(* Logix 5000 project; controller Safety vendor 1 type 14 code 86 rev 19.11; software revision 19.01; part 7 of 17 *)
(* tags used below, declared in another part *)
   ToCitect4 : DINT[64];   // (To Citect4)
   x172CR460 : ALIAS FOR SDPLC:1:I.Pt00Data;   // Shear Die Drive Main Contactor Safety Relay Input
   x172CR510 : ALIAS FOR SDPLC:1:I.Pt01Data;   // Shear Die Drive Enable Safety Relay Input
   x533PB470a : ALIAS FOR H1:6:I.Pt00Data;   // Sheeter Emergency Stop Pushbutton
   x533PB470b : ALIAS FOR H1:6:I.Pt01Data;   // Sheeter Emergency Stop Pushbutton
   x702MTR191FF : ALIAS FOR MCC1:1:I.Pt00Data;   // Rewind Pinch Roll Fwd Fdbk
   x702MTR191RF : ALIAS FOR MCC1:1:I.Pt01Data;   // Rewind Pinch Roll Rev Fdbk
   x708MTR080FF : ALIAS FOR MCC1:1:I.Pt04Data;   // Flattener Drive Motor Fwd Fdbk
   x708MTR080RF : ALIAS FOR MCC1:1:I.Pt05Data;   // Flattener Drive Motor Rev Fdbk
   x708MTR250FF : ALIAS FOR MCC1:1:I.Pt06Data;   // Unwind Holddown Roll Drive Motor Fwd Fdbk
   x708MTR250RF : ALIAS FOR MCC1:1:I.Pt07Data;   // Unwind Holddown Roll Drive Motor Rev Fdbk
   x753MTR190FF : ALIAS FOR MCC3:1:I.Pt00Data;   // Trimmer Pinch Roll Fwd Fdbk
   x753MTR190RF : ALIAS FOR MCC3:1:I.Pt01Data;   // Trimmer Pinch Roll Rev Fdbk
   x759MTR080SE : ALIAS FOR MCC3:4:O.Pt02Data;   // Scrap Choppers Width Adjust Safety Enable
   x759MTR080SP : ALIAS FOR MCC3:4:O.Pt01Data;   // Scrap Choppers Width Adjust Safety Power
   x761MTR081RF : ALIAS FOR MCC3:1:I.Pt02Data;   // Trimmer Scrap Conveyor RunFdbk
   x778MTR080RF : ALIAS FOR MCC4:1:I.Pt00Data;   // Shear Crank Motor Run Fdbk
   x802MTR080FF : ALIAS FOR MCC5:1:I.Pt00Data;   // Stacker Side Guide Lift Fwd Fdbk/Up
   x802MTR080RF : ALIAS FOR MCC5:1:I.Pt01Data;   // Stacker Side Guide Lift Rev Fdbk/Down
   x802MTR230FF : ALIAS FOR MCC5:1:I.Pt02Data;   // Scrap Horizontal Conveyor Run Fwd Fdbk
   x802MTR230RF : ALIAS FOR MCC5:1:I.Pt03Data;   // Scrap Horizontal Conveyor Run Rev Fdbk
   x802MTR231FF : ALIAS FOR MCC5:1:I.Pt04Data;   // Stacker Chain Fwd Fdbk
   x802MTR231RF : ALIAS FOR MCC5:1:I.Pt05Data;   // Stacker Chain Rev Fdbk
   y172CR460 : ALIAS FOR SDPLC:2:O.Pt00Data;   // Shear Die Drive Main Contactor Safety Relay Output
   y172CR510 : ALIAS FOR SDPLC:2:O.Pt01Data;   // Shear Die Drive Enable Safety Relay Output
   y172CR550 : ALIAS FOR SDPLC:2:O.Pt02Data;   // Line Soleniod Safe-Off
   y702MTR191FC : ALIAS FOR MCC1:6:O.Pt00Data;   // Rewind Pinch Roll Fwd Cmd
   y702MTR191RC : ALIAS FOR MCC1:6:O.Pt01Data;   // Rewind Pinch Roll Rev Cmd
   y708MTR080FC : ALIAS FOR MCC1:6:O.Pt04Data;   // Flattener Drive Motor Fwd Cmd
   y708MTR080RC : ALIAS FOR MCC1:6:O.Pt05Data;   // Flattener Drive Motor Rev Cmd
   y708MTR250FC : ALIAS FOR MCC1:6:O.Pt06Data;   // Unwind Holddown Roll Drive Motor Fwd Cmd
   y708MTR250RC : ALIAS FOR MCC1:6:O.Pt07Data;   // Unwind Holddown Roll Drive Motor Rev Cmd
   y725MTR080SE : ALIAS FOR MCC2:1:O.Pt01Data;   // Unwind Pinch Roll Safety Enable
   y725MTR080SP : ALIAS FOR MCC2:1:O.Pt00Data;   // Unwind Pinch Roll Safety Power
   y727MTR080SE : ALIAS FOR MCC2:1:O.Pt05Data;   // Paper Winder Safety Enable
   y727MTR080SP : ALIAS FOR MCC2:1:O.Pt04Data;   // Paper Winder Safety Power
   y729MTR080SE : ALIAS FOR MCC2:1:O.Pt03Data;   // Washtank Pinch Roll 4 Safety Enable
   y729MTR080SP : ALIAS FOR MCC2:1:O.Pt02Data;   // Washtank Pinch Roll 4 Safety Power
   y731MTR080SE : ALIAS FOR MCC2:1:O.Pt07Data;   // Washtank Pinch Roll 1 Safety Enable
   y731MTR080SP : ALIAS FOR MCC2:1:O.Pt06Data;   // Washtank Pinch Roll 1 Safety Power
   y733MTR080SE : ALIAS FOR MCC2:2:O.Pt01Data;   // Washtank Pinch Roll 2 Safety Enable
   y733MTR080SP : ALIAS FOR MCC2:2:O.Pt00Data;   // Washtank Pinch Roll 2 Safety Power
   y735MTR080SE : ALIAS FOR MCC2:2:O.Pt03Data;   // Washtank Pinch Roll 3 Safety Enable
   y735MTR080SP : ALIAS FOR MCC2:2:O.Pt02Data;   // Washtank Pinch Roll 3 Safety Power
   y751MTR080SE : ALIAS FOR MCC3:3:O.Pt04Data;   // Trimmer Knives Safety Enable
   y751MTR080SP : ALIAS FOR MCC3:3:O.Pt03Data;   // Trimmer Knives Safety Power
   y753MTR190FC : ALIAS FOR MCC3:3:O.Pt00Data;   // Trimmer Pinch Roll Fwd Cmd
   y753MTR190RC : ALIAS FOR MCC3:3:O.Pt01Data;   // Trimmer Pinch Roll Rev Cmd
   y754MTR080SE : ALIAS FOR MCC3:3:O.Pt06Data;   // Side Guide Width Adjust Safety Enable
   y754MTR080SP : ALIAS FOR MCC3:3:O.Pt05Data;   // Side Guide Width Adjust Safety Power
   y755MTR080SE : ALIAS FOR MCC3:4:O.Pt00Data;   // Trimmer Knives Width Adjust Safety Enable
   y755MTR080SP : ALIAS FOR MCC3:3:O.Pt07Data;   // Trimmer Knives Width Adjust Safety Power
   y761MTR081RC : ALIAS FOR MCC3:3:O.Pt02Data;   // Trimmer Scrap Conveyor RunCmd
   y762MTR080SE : ALIAS FOR MCC3:4:O.Pt04Data;   // Scrap Choppers Safety Enable
   y762MTR080SP : ALIAS FOR MCC3:4:O.Pt03Data;   // Scrap Choppers Safety Power
   y776MTR080SE : ALIAS FOR MCC4:3:O.Pt07Data;   // Shear Metering Backup Roll Safety Enable
   y776MTR080SP : ALIAS FOR MCC4:3:O.Pt06Data;   // Shear Metering Backup Roll Safety Power
   y778MTR080RC : ALIAS FOR MCC4:4:O.Pt00Data;   // Shear Die Crank Run Cmd
   y779MTR080SE : ALIAS FOR MCC4:3:O.Pt01Data;   // Shear Pinch Roll Safety Enable
   y779MTR080SP : ALIAS FOR MCC4:3:O.Pt00Data;   // Shear Pinch Roll Safety Power
   y782MTR080SE : ALIAS FOR MCC4:3:O.Pt03Data;   // Sheeter Pinch Roll Safety Enable
   y782MTR080SP : ALIAS FOR MCC4:3:O.Pt02Data;   // Sheeter Pinch Roll Safety Power
   y785MTR080SE : ALIAS FOR MCC4:3:O.Pt05Data;   // Stacker Blower Safety Enable
   y785MTR080SP : ALIAS FOR MCC4:3:O.Pt04Data;   // Stacker Blower Safety Power
   y800MTR080SE : ALIAS FOR MCC5:3:O.Pt01Data;   // Scrap Incline Conveyor Safety Enable
   y800MTR080SP : ALIAS FOR MCC5:3:O.Pt00Data;   // Scrap Incline Conveyor Safety Power
   y802MTR080FC : ALIAS FOR MCC5:4:O.Pt04Data;   // Stacker Side Guide Lift Fwd Cmd/Up
   y802MTR080RC : ALIAS FOR MCC5:4:O.Pt05Data;   // Stacker Side Guide Lift Rev Cmd/Down
   y802MTR230FC : ALIAS FOR MCC5:4:O.Pt06Data;   // Scrap Horizontal Conveyor Fwd Cmd
   y802MTR230RC : ALIAS FOR MCC5:4:O.Pt07Data;   // Scrap Horizontal Conveyor Rev Cmd
   y802MTR231FC : ALIAS FOR MCC5:5:O.Pt00Data;   // Stacker Chain Fwd Cmd
   y802MTR231RC : ALIAS FOR MCC5:5:O.Pt01Data;   // Stacker Chain Rev Cmd
   y804MTR080SE : ALIAS FOR MCC5:3:O.Pt03Data;   // Stacker Back Stop Safety Enable
   y804MTR080SP : ALIAS FOR MCC5:3:O.Pt02Data;   // Stacker Back Stop Safety Power
   y806MTR080SE : ALIAS FOR MCC5:3:O.Pt05Data;   // Product Conveyor 3 Safety Enable
   y806MTR080SP : ALIAS FOR MCC5:3:O.Pt04Data;   // Product Conveyor 3 Safety Power
   y808MTR080SE : ALIAS FOR MCC5:3:O.Pt07Data;   // Product Conveyor 1 Safety Enable
   y808MTR080SP : ALIAS FOR MCC5:3:O.Pt06Data;   // Product Conveyor 1 Safety Power
   y810MTR080SE : ALIAS FOR MCC5:4:O.Pt01Data;   // Product Conveyor 2 Safety Enable
   y810MTR080SP : ALIAS FOR MCC5:4:O.Pt00Data;   // Product Conveyor 2 Safety Power
   y812MTR080SE : ALIAS FOR MCC5:4:O.Pt03Data;   // Shear Conveyor Safety Enable
   y812MTR080SP : ALIAS FOR MCC5:4:O.Pt02Data;   // Shear Conveyor Safety Power
(* Comms, continued *)

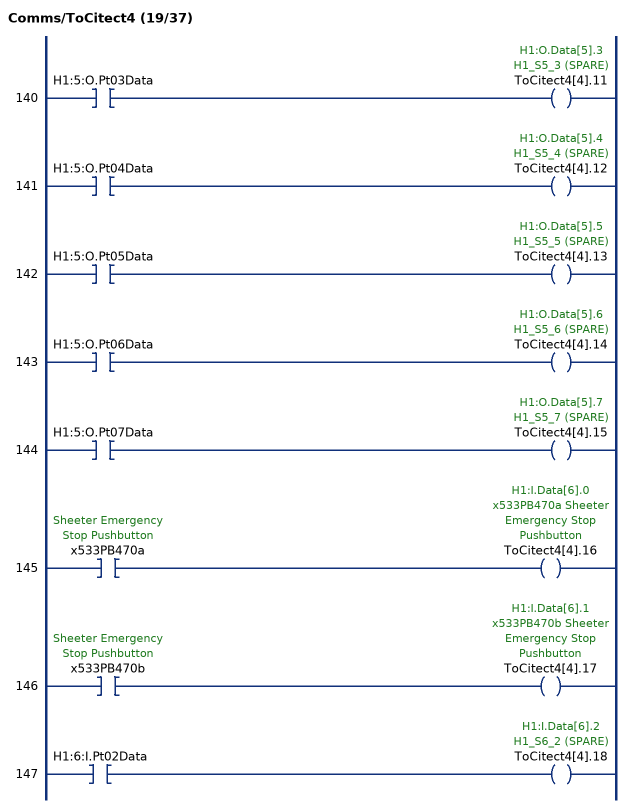
   140: XIC(H1:5:O.Pt03Data)OTE(ToCitect4[4].11);
   141: XIC(H1:5:O.Pt04Data)OTE(ToCitect4[4].12);
   142: XIC(H1:5:O.Pt05Data)OTE(ToCitect4[4].13);
   143: XIC(H1:5:O.Pt06Data)OTE(ToCitect4[4].14);
   144: XIC(H1:5:O.Pt07Data)OTE(ToCitect4[4].15);
   145: XIC(x533PB470a)OTE(ToCitect4[4].16);
   146: XIC(x533PB470b)OTE(ToCitect4[4].17);
   147: XIC(H1:6:I.Pt02Data)OTE(ToCitect4[4].18);
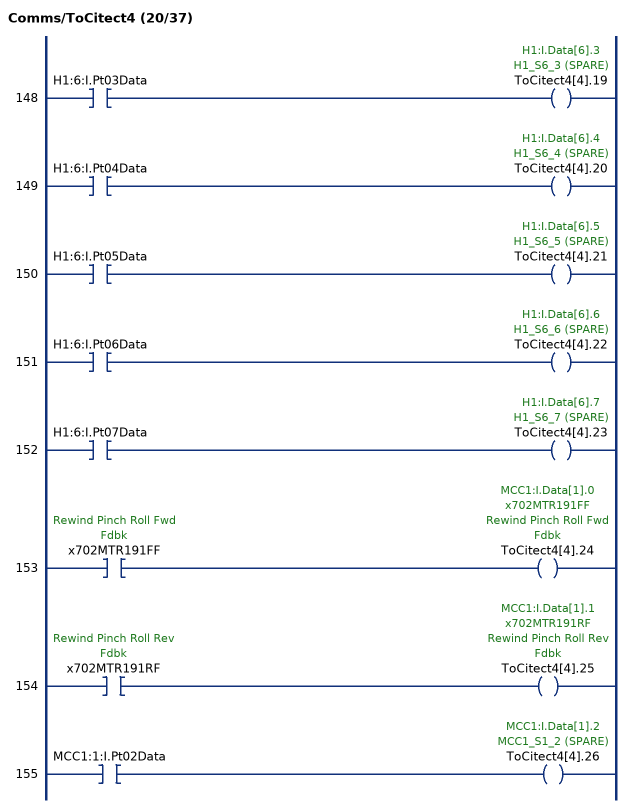
   148: XIC(H1:6:I.Pt03Data)OTE(ToCitect4[4].19);
   149: XIC(H1:6:I.Pt04Data)OTE(ToCitect4[4].20);
   150: XIC(H1:6:I.Pt05Data)OTE(ToCitect4[4].21);
   151: XIC(H1:6:I.Pt06Data)OTE(ToCitect4[4].22);
   152: XIC(H1:6:I.Pt07Data)OTE(ToCitect4[4].23);
   153: XIC(x702MTR191FF)OTE(ToCitect4[4].24);
   154: XIC(x702MTR191RF)OTE(ToCitect4[4].25);
   155: XIC(MCC1:1:I.Pt02Data)OTE(ToCitect4[4].26);
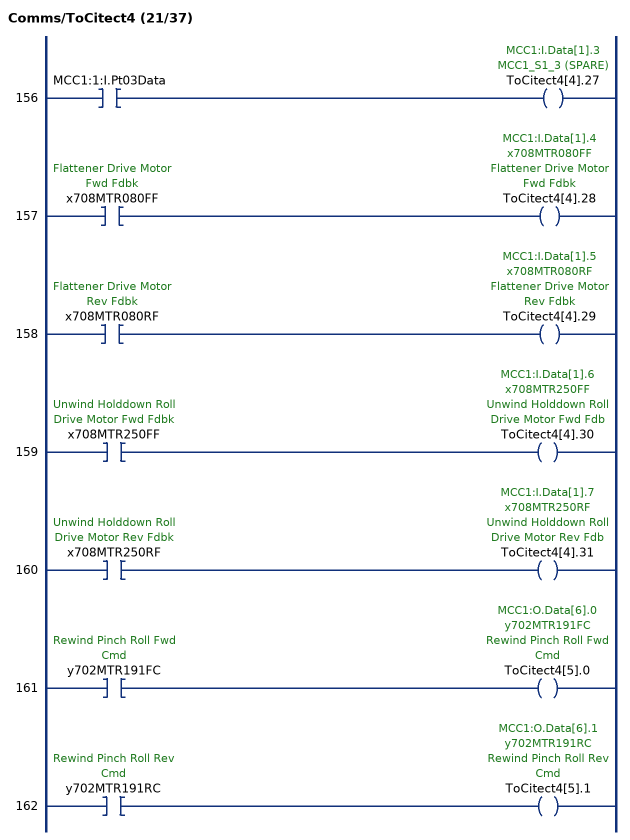
   156: XIC(MCC1:1:I.Pt03Data)OTE(ToCitect4[4].27);
   157: XIC(x708MTR080FF)OTE(ToCitect4[4].28);
   158: XIC(x708MTR080RF)OTE(ToCitect4[4].29);
   159: XIC(x708MTR250FF)OTE(ToCitect4[4].30);
   160: XIC(x708MTR250RF)OTE(ToCitect4[4].31);
   161: XIC(y702MTR191FC)OTE(ToCitect4[5].0);
   162: XIC(y702MTR191RC)OTE(ToCitect4[5].1);
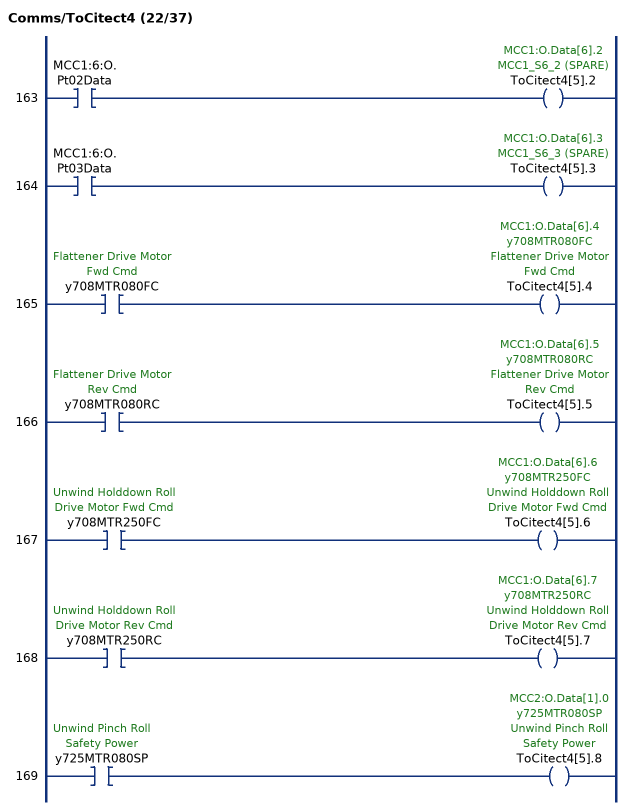
   163: XIC(MCC1:6:O.Pt02Data)OTE(ToCitect4[5].2);
   164: XIC(MCC1:6:O.Pt03Data)OTE(ToCitect4[5].3);
   165: XIC(y708MTR080FC)OTE(ToCitect4[5].4);
   166: XIC(y708MTR080RC)OTE(ToCitect4[5].5);
   167: XIC(y708MTR250FC)OTE(ToCitect4[5].6);
   168: XIC(y708MTR250RC)OTE(ToCitect4[5].7);
   169: XIC(y725MTR080SP)OTE(ToCitect4[5].8);
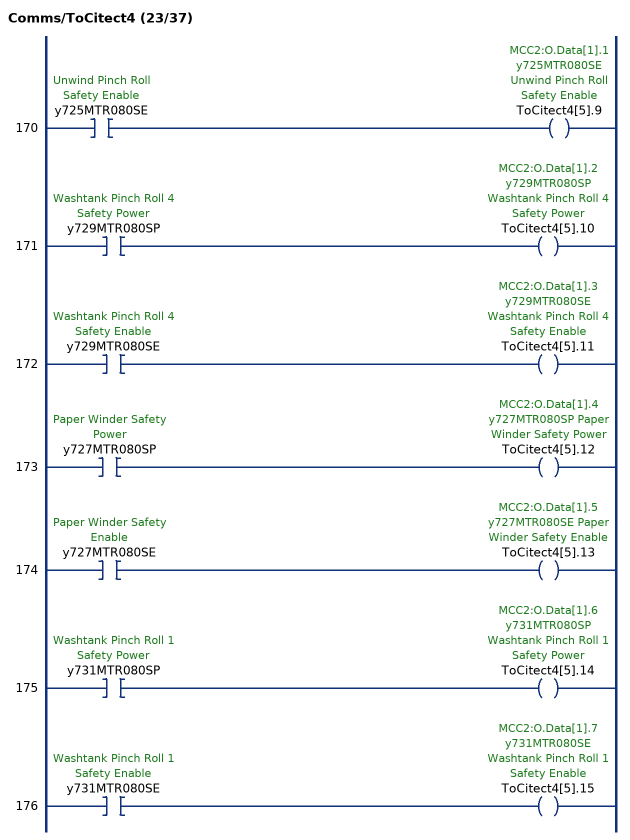
   170: XIC(y725MTR080SE)OTE(ToCitect4[5].9);
   171: XIC(y729MTR080SP)OTE(ToCitect4[5].10);
   172: XIC(y729MTR080SE)OTE(ToCitect4[5].11);
   173: XIC(y727MTR080SP)OTE(ToCitect4[5].12);
   174: XIC(y727MTR080SE)OTE(ToCitect4[5].13);
   175: XIC(y731MTR080SP)OTE(ToCitect4[5].14);
   176: XIC(y731MTR080SE)OTE(ToCitect4[5].15);
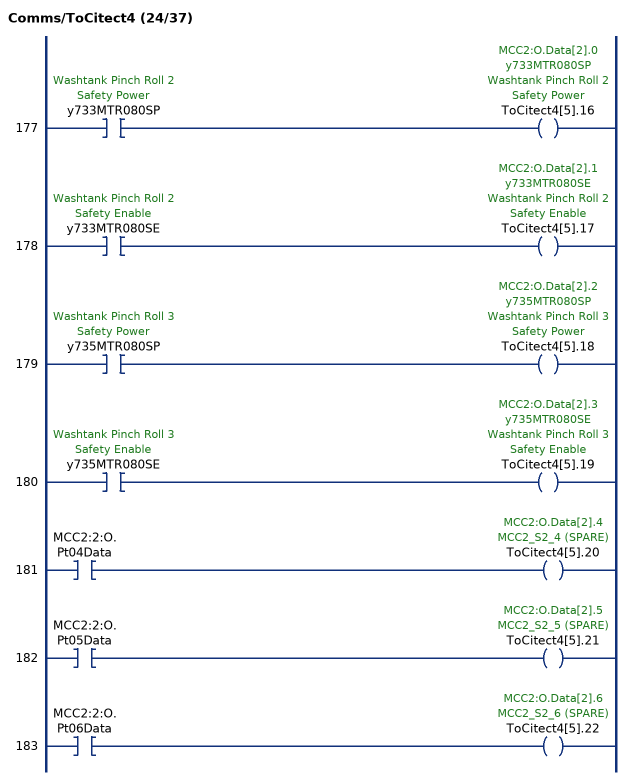
   177: XIC(y733MTR080SP)OTE(ToCitect4[5].16);
   178: XIC(y733MTR080SE)OTE(ToCitect4[5].17);
   179: XIC(y735MTR080SP)OTE(ToCitect4[5].18);
   180: XIC(y735MTR080SE)OTE(ToCitect4[5].19);
   181: XIC(MCC2:2:O.Pt04Data)OTE(ToCitect4[5].20);
   182: XIC(MCC2:2:O.Pt05Data)OTE(ToCitect4[5].21);
   183: XIC(MCC2:2:O.Pt06Data)OTE(ToCitect4[5].22);
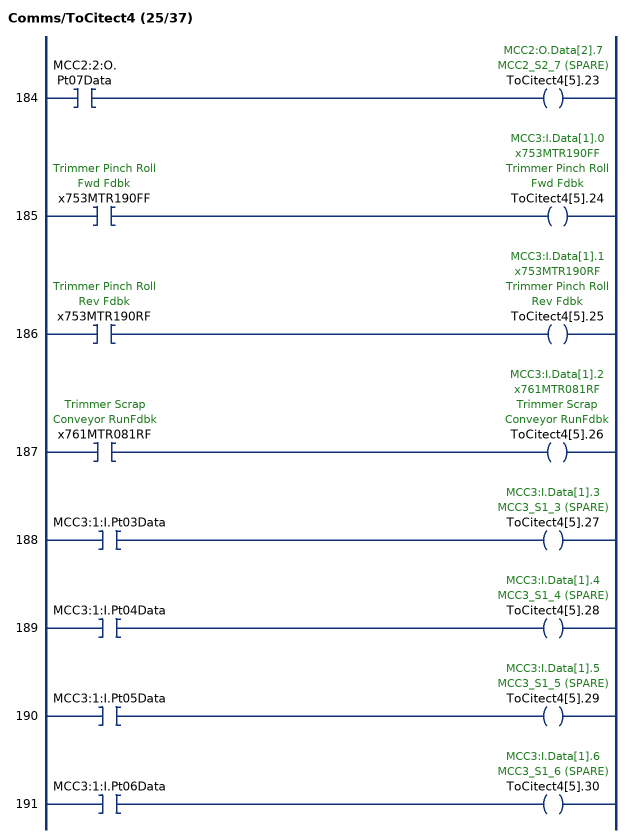
   184: XIC(MCC2:2:O.Pt07Data)OTE(ToCitect4[5].23);
   185: XIC(x753MTR190FF)OTE(ToCitect4[5].24);
   186: XIC(x753MTR190RF)OTE(ToCitect4[5].25);
   187: XIC(x761MTR081RF)OTE(ToCitect4[5].26);
   188: XIC(MCC3:1:I.Pt03Data)OTE(ToCitect4[5].27);
   189: XIC(MCC3:1:I.Pt04Data)OTE(ToCitect4[5].28);
   190: XIC(MCC3:1:I.Pt05Data)OTE(ToCitect4[5].29);
   191: XIC(MCC3:1:I.Pt06Data)OTE(ToCitect4[5].30);
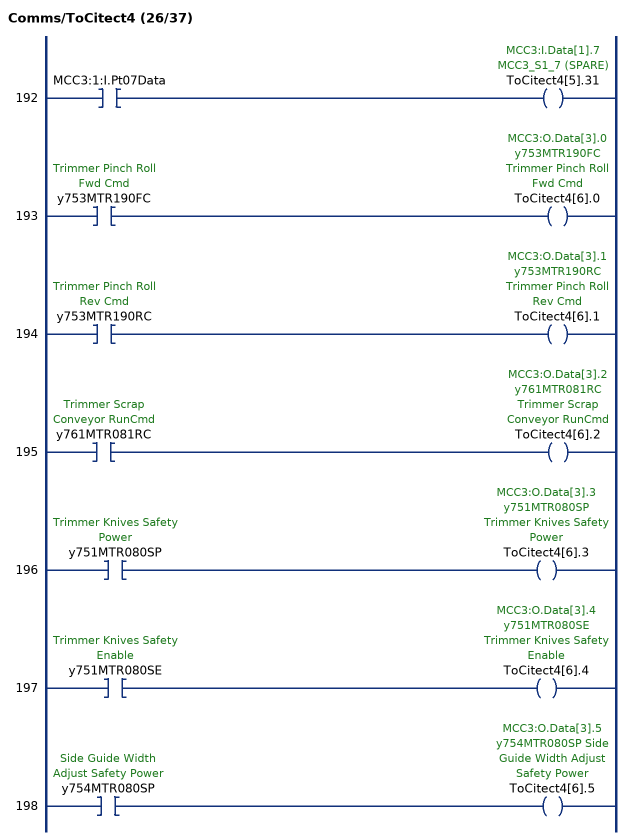
   192: XIC(MCC3:1:I.Pt07Data)OTE(ToCitect4[5].31);
   193: XIC(y753MTR190FC)OTE(ToCitect4[6].0);
   194: XIC(y753MTR190RC)OTE(ToCitect4[6].1);
   195: XIC(y761MTR081RC)OTE(ToCitect4[6].2);
   196: XIC(y751MTR080SP)OTE(ToCitect4[6].3);
   197: XIC(y751MTR080SE)OTE(ToCitect4[6].4);
   198: XIC(y754MTR080SP)OTE(ToCitect4[6].5);
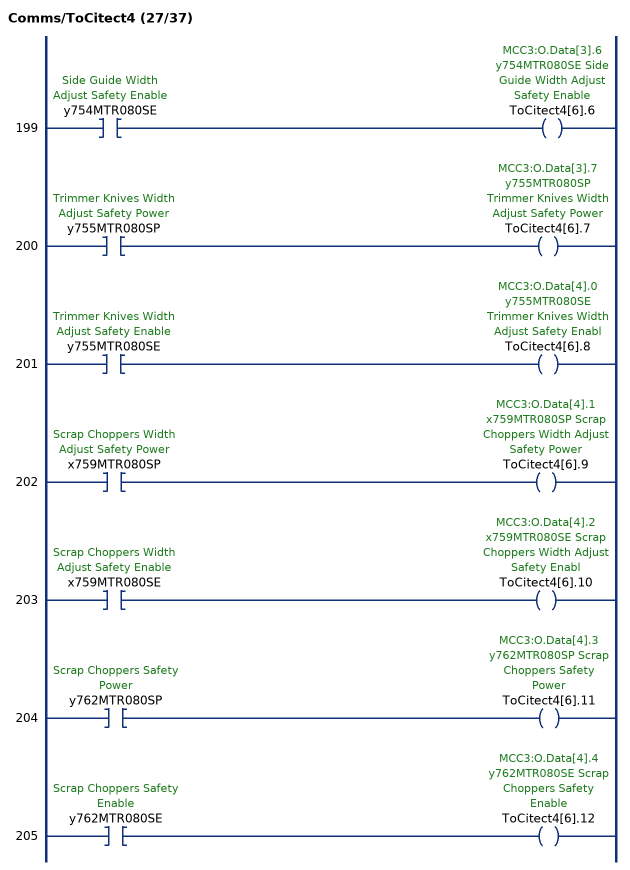
   199: XIC(y754MTR080SE)OTE(ToCitect4[6].6);
   200: XIC(y755MTR080SP)OTE(ToCitect4[6].7);
   201: XIC(y755MTR080SE)OTE(ToCitect4[6].8);
   202: XIC(x759MTR080SP)OTE(ToCitect4[6].9);
   203: XIC(x759MTR080SE)OTE(ToCitect4[6].10);
   204: XIC(y762MTR080SP)OTE(ToCitect4[6].11);
   205: XIC(y762MTR080SE)OTE(ToCitect4[6].12);
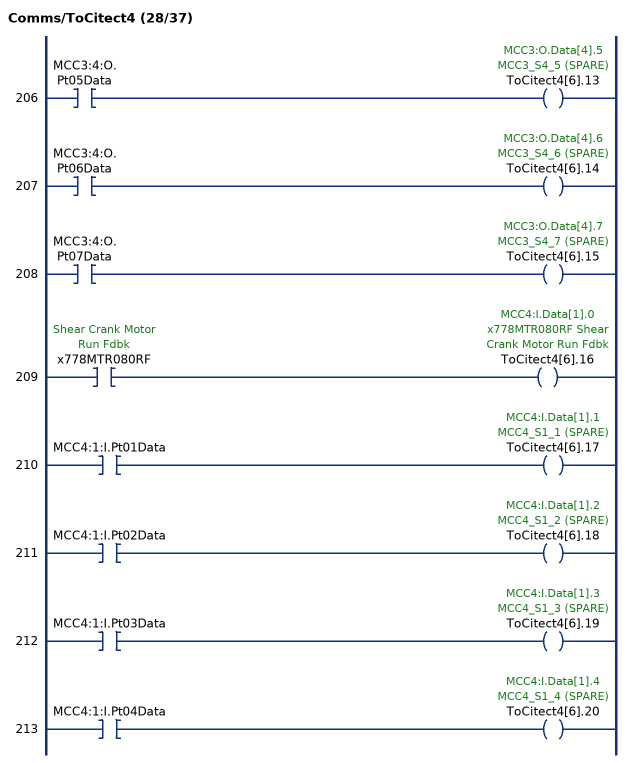
   206: XIC(MCC3:4:O.Pt05Data)OTE(ToCitect4[6].13);
   207: XIC(MCC3:4:O.Pt06Data)OTE(ToCitect4[6].14);
   208: XIC(MCC3:4:O.Pt07Data)OTE(ToCitect4[6].15);
   209: XIC(x778MTR080RF)OTE(ToCitect4[6].16);
   210: XIC(MCC4:1:I.Pt01Data)OTE(ToCitect4[6].17);
   211: XIC(MCC4:1:I.Pt02Data)OTE(ToCitect4[6].18);
   212: XIC(MCC4:1:I.Pt03Data)OTE(ToCitect4[6].19);
   213: XIC(MCC4:1:I.Pt04Data)OTE(ToCitect4[6].20);
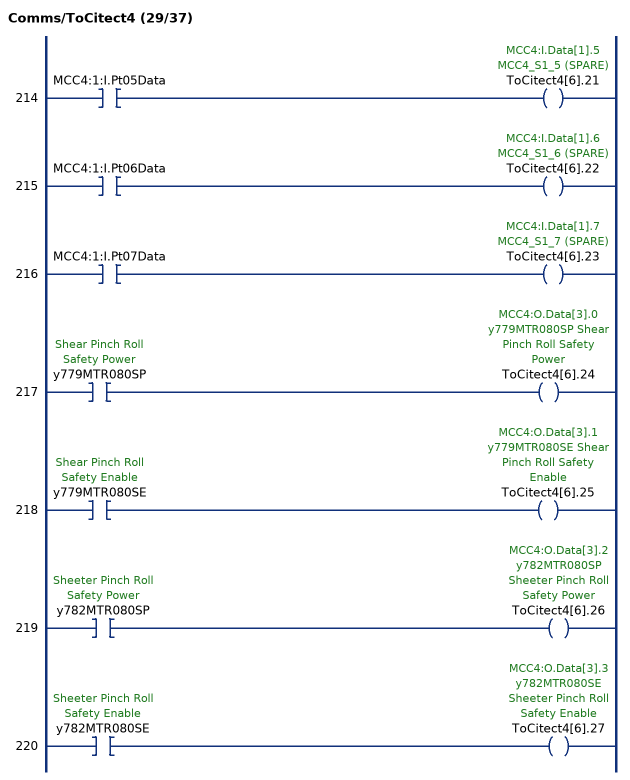
   214: XIC(MCC4:1:I.Pt05Data)OTE(ToCitect4[6].21);
   215: XIC(MCC4:1:I.Pt06Data)OTE(ToCitect4[6].22);
   216: XIC(MCC4:1:I.Pt07Data)OTE(ToCitect4[6].23);
   217: XIC(y779MTR080SP)OTE(ToCitect4[6].24);
   218: XIC(y779MTR080SE)OTE(ToCitect4[6].25);
   219: XIC(y782MTR080SP)OTE(ToCitect4[6].26);
   220: XIC(y782MTR080SE)OTE(ToCitect4[6].27);
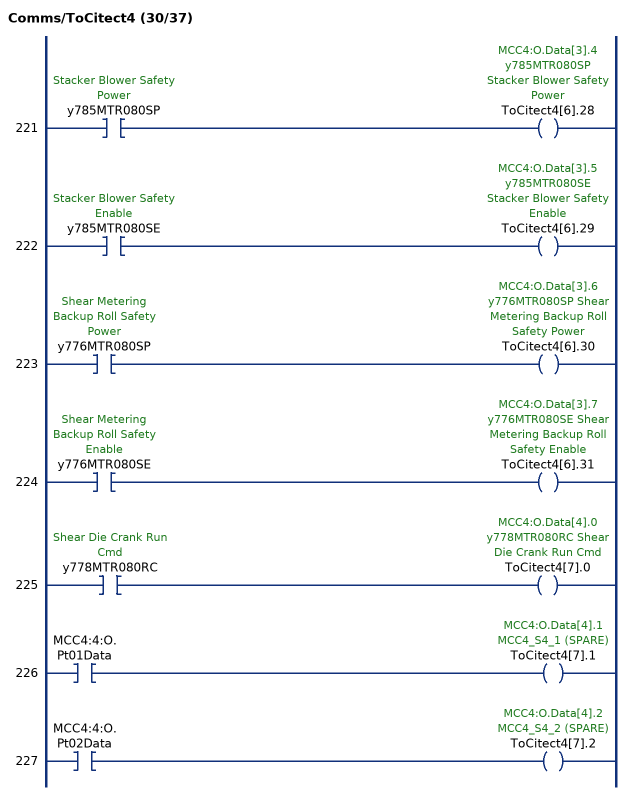
   221: XIC(y785MTR080SP)OTE(ToCitect4[6].28);
   222: XIC(y785MTR080SE)OTE(ToCitect4[6].29);
   223: XIC(y776MTR080SP)OTE(ToCitect4[6].30);
   224: XIC(y776MTR080SE)OTE(ToCitect4[6].31);
   225: XIC(y778MTR080RC)OTE(ToCitect4[7].0);
   226: XIC(MCC4:4:O.Pt01Data)OTE(ToCitect4[7].1);
   227: XIC(MCC4:4:O.Pt02Data)OTE(ToCitect4[7].2);
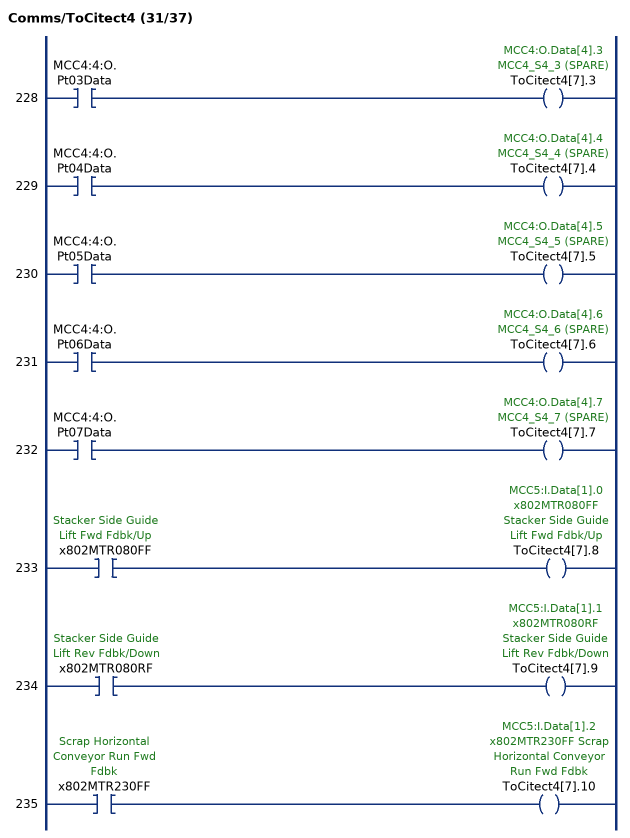
   228: XIC(MCC4:4:O.Pt03Data)OTE(ToCitect4[7].3);
   229: XIC(MCC4:4:O.Pt04Data)OTE(ToCitect4[7].4);
   230: XIC(MCC4:4:O.Pt05Data)OTE(ToCitect4[7].5);
   231: XIC(MCC4:4:O.Pt06Data)OTE(ToCitect4[7].6);
   232: XIC(MCC4:4:O.Pt07Data)OTE(ToCitect4[7].7);
   233: XIC(x802MTR080FF)OTE(ToCitect4[7].8);
   234: XIC(x802MTR080RF)OTE(ToCitect4[7].9);
   235: XIC(x802MTR230FF)OTE(ToCitect4[7].10);
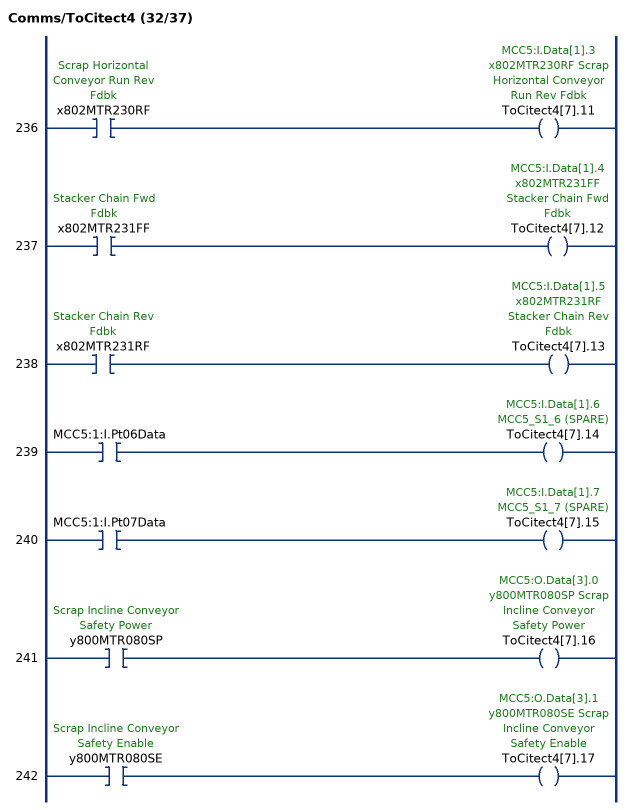
   236: XIC(x802MTR230RF)OTE(ToCitect4[7].11);
   237: XIC(x802MTR231FF)OTE(ToCitect4[7].12);
   238: XIC(x802MTR231RF)OTE(ToCitect4[7].13);
   239: XIC(MCC5:1:I.Pt06Data)OTE(ToCitect4[7].14);
   240: XIC(MCC5:1:I.Pt07Data)OTE(ToCitect4[7].15);
   241: XIC(y800MTR080SP)OTE(ToCitect4[7].16);
   242: XIC(y800MTR080SE)OTE(ToCitect4[7].17);
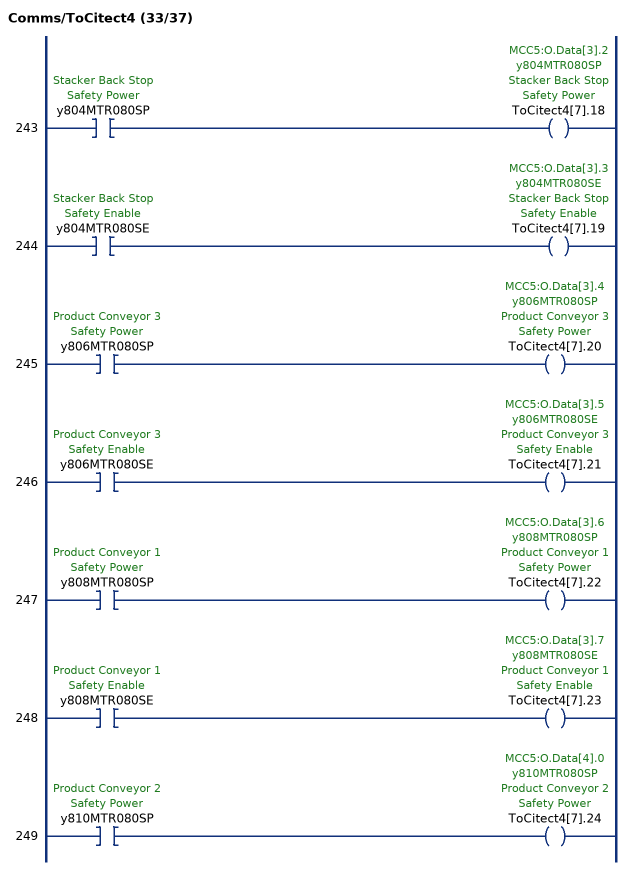
   243: XIC(y804MTR080SP)OTE(ToCitect4[7].18);
   244: XIC(y804MTR080SE)OTE(ToCitect4[7].19);
   245: XIC(y806MTR080SP)OTE(ToCitect4[7].20);
   246: XIC(y806MTR080SE)OTE(ToCitect4[7].21);
   247: XIC(y808MTR080SP)OTE(ToCitect4[7].22);
   248: XIC(y808MTR080SE)OTE(ToCitect4[7].23);
   249: XIC(y810MTR080SP)OTE(ToCitect4[7].24);
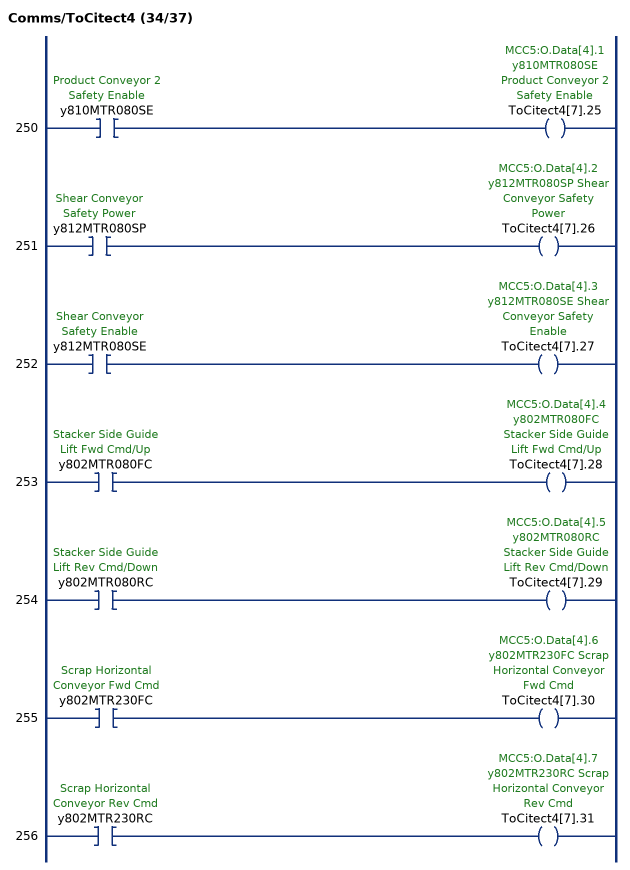
   250: XIC(y810MTR080SE)OTE(ToCitect4[7].25);
   251: XIC(y812MTR080SP)OTE(ToCitect4[7].26);
   252: XIC(y812MTR080SE)OTE(ToCitect4[7].27);
   253: XIC(y802MTR080FC)OTE(ToCitect4[7].28);
   254: XIC(y802MTR080RC)OTE(ToCitect4[7].29);
   255: XIC(y802MTR230FC)OTE(ToCitect4[7].30);
   256: XIC(y802MTR230RC)OTE(ToCitect4[7].31);
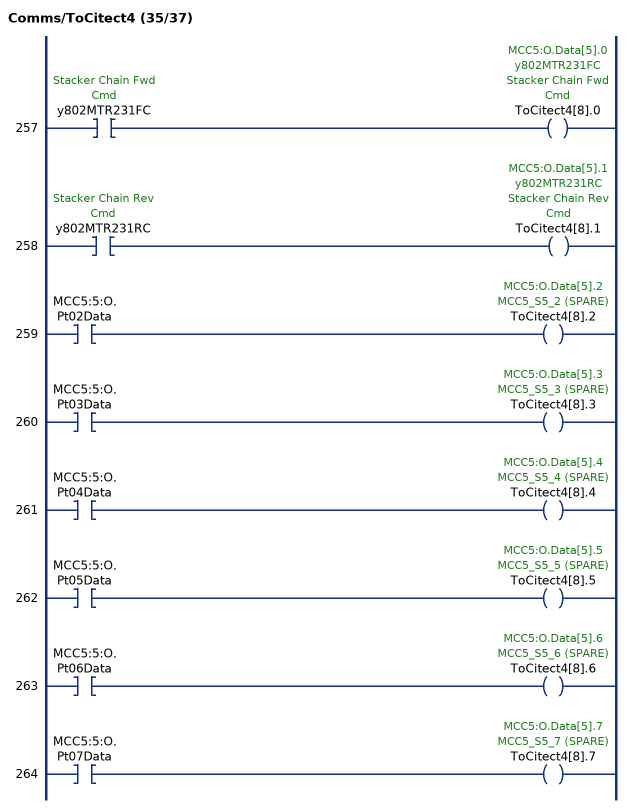
   257: XIC(y802MTR231FC)OTE(ToCitect4[8].0);
   258: XIC(y802MTR231RC)OTE(ToCitect4[8].1);
   259: XIC(MCC5:5:O.Pt02Data)OTE(ToCitect4[8].2);
   260: XIC(MCC5:5:O.Pt03Data)OTE(ToCitect4[8].3);
   261: XIC(MCC5:5:O.Pt04Data)OTE(ToCitect4[8].4);
   262: XIC(MCC5:5:O.Pt05Data)OTE(ToCitect4[8].5);
   263: XIC(MCC5:5:O.Pt06Data)OTE(ToCitect4[8].6);
   264: XIC(MCC5:5:O.Pt07Data)OTE(ToCitect4[8].7);
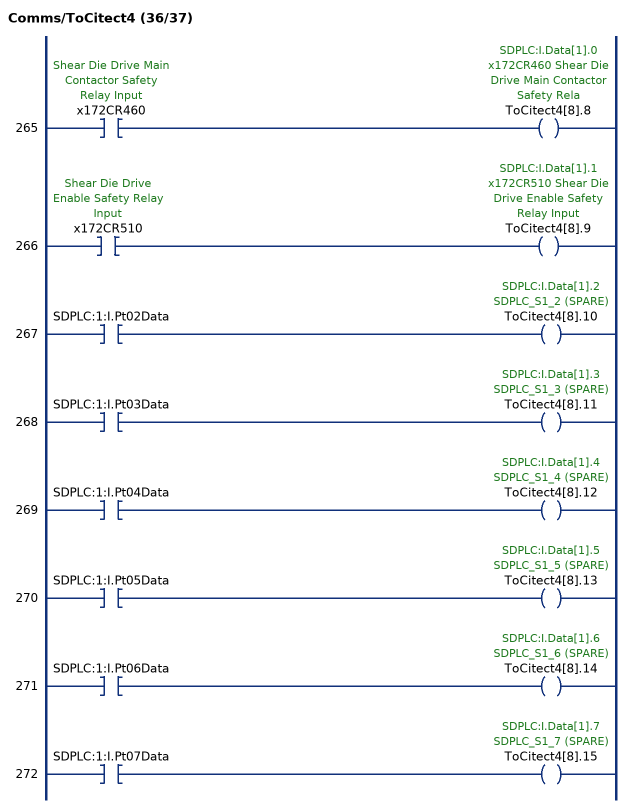
   265: XIC(x172CR460)OTE(ToCitect4[8].8);
   266: XIC(x172CR510)OTE(ToCitect4[8].9);
   267: XIC(SDPLC:1:I.Pt02Data)OTE(ToCitect4[8].10);
   268: XIC(SDPLC:1:I.Pt03Data)OTE(ToCitect4[8].11);
   269: XIC(SDPLC:1:I.Pt04Data)OTE(ToCitect4[8].12);
   270: XIC(SDPLC:1:I.Pt05Data)OTE(ToCitect4[8].13);
   271: XIC(SDPLC:1:I.Pt06Data)OTE(ToCitect4[8].14);
   272: XIC(SDPLC:1:I.Pt07Data)OTE(ToCitect4[8].15);
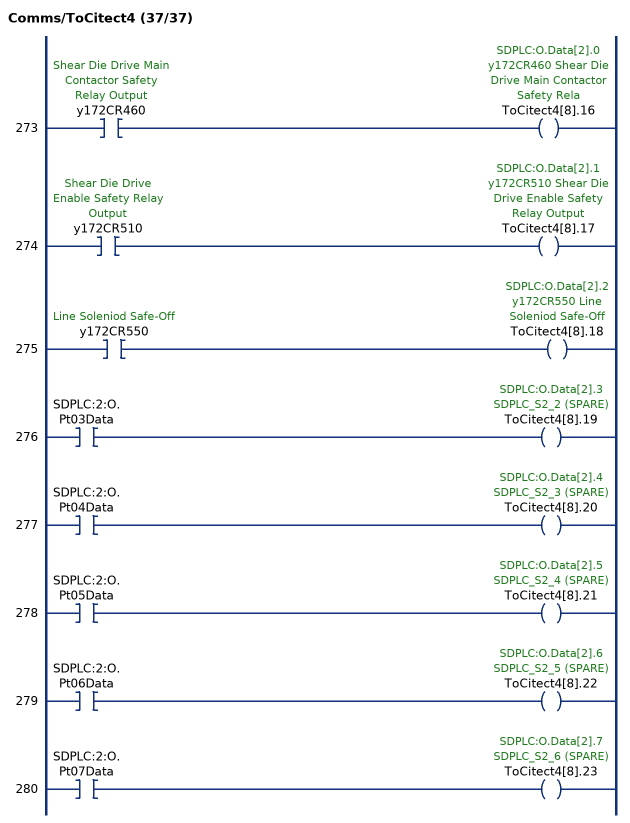
   273: XIC(y172CR460)OTE(ToCitect4[8].16);
   274: XIC(y172CR510)OTE(ToCitect4[8].17);
   275: XIC(y172CR550)OTE(ToCitect4[8].18);
   276: XIC(SDPLC:2:O.Pt03Data)OTE(ToCitect4[8].19);
   277: XIC(SDPLC:2:O.Pt04Data)OTE(ToCitect4[8].20);
   278: XIC(SDPLC:2:O.Pt05Data)OTE(ToCitect4[8].21);
   279: XIC(SDPLC:2:O.Pt06Data)OTE(ToCitect4[8].22);
   280: XIC(SDPLC:2:O.Pt07Data)OTE(ToCitect4[8].23);
END_ROUTINE
END_PROGRAM
